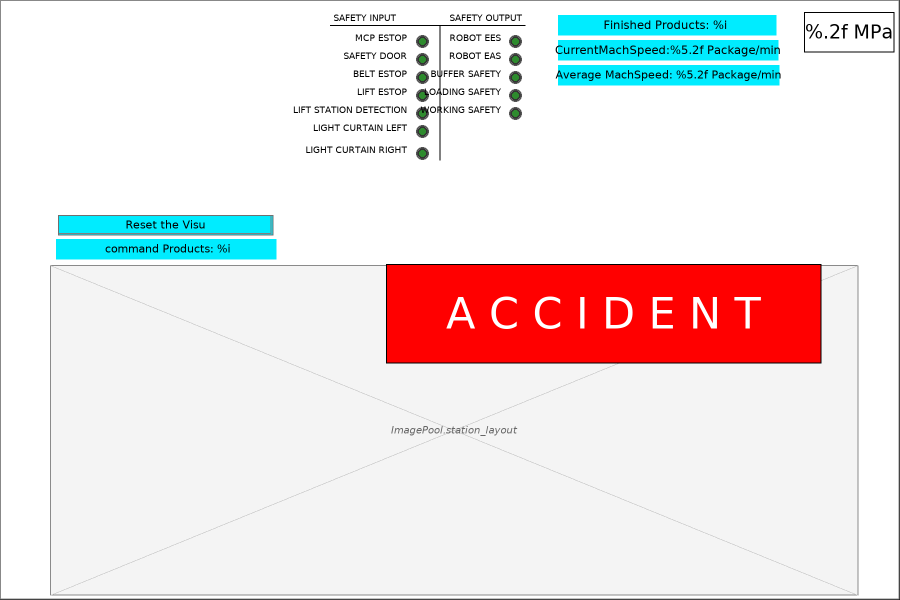
VISUALIZATION VIS_TemplateMachine  // 900x600
    Rectangle (0,0 900x600)
    Image (50,265 808x330), image: ImagePool.station_layout
    Rectangle (386,264 435x99), "A C C I D E N T", invisible if: NOT (MAIN.application.tote_subsystem.status=MachineStatus.ERROR)
    Rectangle (56,239 220x20), "command Products: %i", text variable: GVL.PackTags.Command.Parameter[1].Value, colour toggle: (MAIN.fbVisu.bInValidEntry OR GVL.PackTags.Admin.Warning[1].Trigger), invisible if: NOT ( MAIN.fbMachine.eMode = 1)
        OnMouseClick: write GVL.nVisuProductCommand via Default
    Rectangle (558,15 218x20), "Finished Products: %i", text variable: GVL.PackTags.Admin.ProdProcessedCount[1].Count, invisible if: NOT ( MAIN.fbMachine.eMode = 1)
    Button (58,215 215x20), "Reset the Visu", invisible if: (MAIN.fbMachine.eMode = 1 AND (MAIN.fbMachine.eState = ePMLState_Clearing OR MAIN.fbMachine.eState = ePMLState_Aborting OR MAIN.fbMachine.eState = ePMLState_Stopping OR MAIN.fbMachine.eState = ePMLState_Resetting OR MAIN.fbMachine.eState = ePMLState_Starting OR MAIN.fbMachine.eState = ePMLState_Execute OR MAIN.fbMachine.eState = ePMLState_Completing OR MAIN.fbMachine.eState = ePMLState_Suspending OR MAIN.fbMachine.eState = ePMLState_Holding))
        tap GVL.stChangeIntoProduction.bYesReset
    Rectangle (558,40 220x20), "CurrentMachSpeed:%5.2f Package/min", text variable: GVL.PackTags.Status.CurMachineSpeed, invisible if: NOT ( MAIN.fbMachine.eMode = 1)
    Rectangle (558,65 221x20), "Average MachSpeed: %5.2f Package/min", text variable: GVL.PackTags.Status.MachineSpeed, invisible if: NOT ( MAIN.fbMachine.eMode = 1)
    Lamp1 (415,34 15x15), variable: MAIN.application.safety.mcp_estop, style: Lamp-Lamp1-Green
    Label (330,34 80x8), "MCP ESTOP"
    Lamp1 (415,70 15x15), variable: MAIN.application.safety.belt_estop, style: Lamp-Lamp1-Green
    Label (330,70 80x8), "BELT ESTOP"
    Lamp1 (415,88 15x15), variable: MAIN.application.safety.lift_estop, style: Lamp-Lamp1-Green
    Label (330,88 80x8), "LIFT ESTOP"
    Lamp1 (415,106 15x15), variable: MAIN.application.safety.lift_station_detection, style: Lamp-Lamp1-Green
    Label (330,106 80x8), "LIFT STATION DETECTION"
    Lamp1 (415,52 15x15), variable: MAIN.application.safety.mcp_safetyDoor, style: Lamp-Lamp1-Green
    Label (330,52 80x8), "SAFETY DOOR"
    Lamp1 (415,124 15x15), variable: MAIN.application.safety.lift_lightCurtain_left, style: Lamp-Lamp1-Green
    Label (330,124 80x8), "LIGHT CURTAIN LEFT"
    Lamp1 (415,146 15x15), variable: MAIN.application.safety.lift_lightCurtain_right, style: Lamp-Lamp1-Green
    Label (330,146 80x8), "LIGHT CURTAIN RIGHT"
    Lamp1 (508,34 15x15), variable: MAIN.application.safety.robot_EES, style: Lamp-Lamp1-Green
    Label (444,34 60x8), "ROBOT EES"
    Lamp1 (508,70 15x15), variable: MAIN.application.safety.buffer_safety, style: Lamp-Lamp1-Green
    Label (444,70 60x8), "BUFFER SAFETY"
    Lamp1 (508,88 15x15), variable: MAIN.application.safety.loading_safety, style: Lamp-Lamp1-Green
    Label (444,88 60x8), "LOADING SAFETY"
    Lamp1 (508,106 15x15), variable: MAIN.application.safety.working_safety, style: Lamp-Lamp1-Green
    Label (444,106 60x8), "WORKING SAFETY"
    Lamp1 (508,52 15x15), variable: MAIN.application.safety.robot_EAS, style: Lamp-Lamp1-Green
    Label (444,52 60x8), "ROBOT EAS"
    Line (440,160) (440,25)
    Label (315,12 100x12), "SAFETY INPUT"
    Label (436,12 100x12), "SAFETY OUTPUT"
    Line (330,25) (525,25)
    Rectangle (804,12 90x40), "%.2f MPa", text variable: MAIN.application.air_pressure_subsystem.current_air_pressure
END_VISUALIZATION

(* stored: Version 1.1.0.1, ProductVersion 3.1.4024.12
   Visu VIS_TemplateMachine: Id {9421e918-9a93-4f23-9733-2bf87c96933b} *)
